FUNCTION_BLOCK CU030ExampleCompositComponent EXTENDS TcoCore.TcoComponent
VAR_INPUT
END_VAR
VAR_OUTPUT
END_VAR
VAR
END_VAR

END_FUNCTION_BLOCK

(* stored: Version 1.1.0.1
   POU CU030ExampleCompositComponent: Id {2caa1da1-ca95-4d44-9c56-e0204ef86c62}, SpecialFunc None *)
